# B&R Automation Studio project FactoryIO_Storage
Automation Studio 4.12.2.93; technology packages: mappView 5.16.1

## Configuration Config1

CPU PC_any, AutomationRuntime B4.93, Build 4.1.2, Vc V4.72.6

### Task classes (Cpu.sw)
```
Cyclic#1 (cycle 20000 us):
  _1000_SCTR <- _1000_SCTRL.prg
  _1100_CSYS <- _1100_CSYS.prg
  _1500_PPS <- _1500_PPS.prg
  _1700_HMI <- _1700_HMI.prg
  _1600_SSYS <- _1600_SSYS.prg
  _1400_SRS <- _1400_SRS.prg
  _1300_CS2 <- _1300_CS2.prg
  _1200_CS1 <- _1200_CS1.prg
Binaries: udbdef, FWRules, TCData, sysconf, Role, User, iomap, ashwd, asfw, arconfig, ashwac
Libraries: Library, runtime, astime, asieccon
```

### Hardware
```
OpcUa_any : OpcUa_any v1.0.0.1  [ETH1 -> PC.IF3 [Cable Type=PowerlinkCable, Length=10, Version=1.0.0.3]]
  ServerEndpointUrl = opc.tcp://127.0.0.1:48020
PC : PC_any v1.1.1.0 (OrderNumber=PC)
  ConfigurationID = FactoryIO_Storage_Config1
  Cyclic1Duration = 20000
  FileDevice1
  FileDeviceName1 = USER
  FileDevicePath1 = USER_PATH
  ActivateOpcUa = 1
  OpcUaInformationModels_PV_Version = 1
```

## Logical view

Binary libraries used (declarations not repeated): operator, runtime, astime, AsIecCon

### Global.var - Global variables
```iecst
VAR
	Gv : UDT_Global;
	Opc : UDT_Opc;
END_VAR
```

### Package Logical/Libraries - Global libraries

### Library Logical/Libraries/Library (IEC)

#### Modules.typ - Exported data types
```iecst
TYPE
	UDT_StorageController : 	STRUCT
		Dummy : BOOL;
	END_STRUCT;
	UDT_ControlSystem : 	STRUCT
		Dummy : BOOL;
	END_STRUCT;
	UDT_ConveyorInfeedSystem : 	STRUCT
		ReadyForOffload : BOOL;
	END_STRUCT;
	UDT_ConveyorOutfeedSystem : 	STRUCT
		ReadyForOnload : BOOL;
	END_STRUCT;
	UDT_StorageRackSystem : 	STRUCT
		Dummy : BOOL;
	END_STRUCT;
	UDT_HMI : 	STRUCT
		Dummy : BOOL;
	END_STRUCT;
	UDT_PickAndPlaceSystem : 	STRUCT
		Offloading : UDT_Sequence;
		Loading : UDT_Sequence;
	END_STRUCT;
	UDT_SafetySystem : 	STRUCT
		SafetyStop : BOOL;
		ControlledStop : BOOL;
	END_STRUCT;
END_TYPE
```

#### Library.fun - Exported functions and function blocks
```iecst
{REDUND_ERROR} FUNCTION_BLOCK FB_Loader (*TODO: Add your comment here*) (*$GROUP=User,$CAT=User,$GROUPICON=User.png,$CATICON=User.png*)
	VAR_INPUT
		in_xLimitRight : {REDUND_UNREPLICABLE} BOOL;
		in_xLimitLeft : {REDUND_UNREPLICABLE} BOOL;
		in_xLimitMiddle : {REDUND_UNREPLICABLE} BOOL;
		in_xInterlock : {REDUND_UNREPLICABLE} BOOL;
		in_xMovingX : {REDUND_UNREPLICABLE} BOOL;
		in_xMovingZ : {REDUND_UNREPLICABLE} BOOL;
		in_rZActualPos : REAL;
		in_rXActualPos : REAL;
		in_rLoadDeltaZ : REAL;
		in_xLoadRightReq : BOOL;
		in_xLoadLeftReq : BOOL;
		in_xUnloadRightReq : BOOL;
		in_xUnloadLeftReq : BOOL;
	END_VAR
	VAR_OUTPUT
		out_sStatus : {REDUND_UNREPLICABLE} UDT_Sequence;
		out_xForksLeftOrder : BOOL;
		out_xForksRightOrder : BOOL;
		out_rXSetPoint : REAL;
		out_rZSetPoint : REAL;
		out_xLoaded : BOOL;
	END_VAR
	VAR
		OperateRight : BOOL;
		OperateLeft : BOOL;
		Unload : BOOL;
		Load : BOOL;
		v_InPosition : BOOL;
		v_LoadSequence : DINT;
	END_VAR
END_FUNCTION_BLOCK

{REDUND_ERROR} FUNCTION_BLOCK FB_Crane (*TODO: Add your comment here*) (*$GROUP=User,$CAT=User,$GROUPICON=User.png,$CATICON=User.png*)
	VAR_INPUT
		in_rXSetPointReq : REAL;
		in_rZSetPointReq : REAL;
		in_rZActualPos : REAL;
		in_rXActualPos : REAL;
		in_xInterlock : BOOL;
	END_VAR
	VAR_OUTPUT
		out_sStatus : {REDUND_UNREPLICABLE} UDT_Sequence;
		out_rXSetPoint : REAL;
		out_rZSetPoint : REAL;
	END_VAR
	VAR
		InPosition : BOOL;
		Interlock : BOOL;
		NewRequest : BOOL;
		PreviousXSetPoint : REAL;
		PreviousZSetPoint : REAL;
		FirstScan : BOOL;
	END_VAR
END_FUNCTION_BLOCK
```

#### OPC.typ
```iecst
TYPE
	UDT_OpcInput : 	STRUCT
		StorageController : UDT_StorageControllerInput;
		ControlSystem : UDT_ControlSystemInput;
		ConveyorInfeed : UDT_ConveyorInfeedInput;
		ConveyorOutfeed : UDT_ConveyorOutfeedInput;
		StorageRack : UDT_StorageRackSystemInput;
		PickAndPlace : UDT_PickAndPlaceSystemInput;
		Safety : UDT_SafetySystemInput;
		HMI : UDT_HMIInput;
	END_STRUCT;
	UDT_OpcOutput : 	STRUCT
		StorageController : UDT_StorageControllerOutput;
		ControlSystem : UDT_ControlSystemOutput;
		ConveyorInfeed : UDT_ConveyorInfeedOutput;
		ConveyorOutfeed : UDT_ConveyorOutfeedOutput;
		StorageRack : UDT_StorageRackSystemOutput;
		PickAndPlace : UDT_PickAndPlaceSystemOutput;
		SafetySystem : UDT_SafetySystemOutput;
		HMI : UDT_HMIOutput;
	END_STRUCT;
	UDT_StorageControllerInput : 	STRUCT
		Opc_IO_Factory_Reset : BOOL;
		Opc_IO_Factory_Running : BOOL;
		Opc_IO_Factory_Paused : BOOL;
	END_STRUCT;
	UDT_ControlSystemInput : 	STRUCT
		Opc_IO_StartButton : BOOL;
		Opc_IO_StopButton : BOOL;
		Opc_IO_ManualSwitch : BOOL;
		Opc_IO_AutoSwitch : BOOL;
	END_STRUCT;
	UDT_ConveyorInfeedInput : 	STRUCT
		Opc_IO_AtEntry : BOOL;
		Opc_IO_AtLoad : BOOL;
	END_STRUCT;
	UDT_ConveyorOutfeedInput : 	STRUCT
		Opc_IO_AtExit : BOOL;
		Opc_IO_AtUnload : BOOL;
	END_STRUCT;
	UDT_StorageRackSystemInput : 	STRUCT
		Dummy : BOOL;
	END_STRUCT;
	UDT_PickAndPlaceSystemInput : 	STRUCT
		Opc_IO_PosZ : REAL;
		Opc_IO_PosX : REAL;
		Opc_IO_MovingX : BOOL;
		Opc_IO_MovingZ : BOOL;
		Opc_IO_LeftLimitSwitch : BOOL;
		Opc_IO_RightLimitSwitch : BOOL;
		Opc_IO_MiddleLimitSwitch : BOOL;
	END_STRUCT;
	UDT_SafetySystemInput : 	STRUCT
		Opc_IO_EmergencyStop1 : BOOL;
	END_STRUCT;
	UDT_HMIInput : 	STRUCT
		Dummy : BOOL;
	END_STRUCT;
	UDT_StorageControllerOutput : 	STRUCT
		Dummy : BOOL;
	END_STRUCT;
	UDT_ControlSystemOutput : 	STRUCT
		Opc_IO_ResetLight : BOOL;
		Opc_IO_StopLight : BOOL;
		Opc_IO_StartLight : BOOL;
	END_STRUCT;
	UDT_ConveyorInfeedOutput : 	STRUCT
		Opc_IO_LoadingConveyor : BOOL;
		Opc_IO_EntryConveyor : BOOL;
	END_STRUCT;
	UDT_ConveyorOutfeedOutput : 	STRUCT
		Opc_IO_UnloadConveyor : BOOL;
		Opc_IO_ExitConveyor : BOOL;
	END_STRUCT;
	UDT_StorageRackSystemOutput : 	STRUCT
		Dummy : BOOL;
	END_STRUCT;
	UDT_PickAndPlaceSystemOutput : 	STRUCT
		Opc_IO_ForksRight : BOOL;
		Opc_IO_XAxisSetPoint : REAL;
		Opc_IO_ZAxisSetPoint : REAL;
		Opc_IO_ForksLeft : BOOL;
	END_STRUCT;
	UDT_SafetySystemOutput : 	STRUCT
		Dummy : BOOL;
	END_STRUCT;
	UDT_HMIOutput : 	STRUCT
		Dummy : BOOL;
	END_STRUCT;
END_TYPE
```

#### Global.typ
```iecst
TYPE
	UDT_Opc : 	STRUCT
		In : UDT_OpcInput;
		Out : UDT_OpcOutput;
	END_STRUCT;
	UDT_Global : 	STRUCT
		StorageController : UDT_StorageController;
		ControlSystem : UDT_ControlSystem;
		ConveyorIn : UDT_ConveyorInfeedSystem;
		ConveyorOut : UDT_ConveyorOutfeedSystem;
		StorageRackSystem : UDT_StorageRackSystem;
		HMI : UDT_HMI;
		PickAndPlaceSystem : UDT_PickAndPlaceSystem;
		SafetySystem : UDT_SafetySystem;
	END_STRUCT;
END_TYPE
```

#### States.typ
```iecst
TYPE
	TSystemState :
		(
		Initializing,
		Running,
		Error,
		Maintenance,
		SafetyStop
		);
END_TYPE
```

#### SubState.typ
```iecst
TYPE
	UDT_Sequence : 	STRUCT
		Error : BOOL;
		Idle : BOOL;
		InProgess : BOOL;
		Requested : BOOL;
	END_STRUCT;
END_TYPE
```

#### DataTypes.typ - not listed in the package file held
```iecst
TYPE
	UDT_XYZCoordinate : 	STRUCT
		X : REAL;
		Y : REAL;
		Z : REAL;
	END_STRUCT;

END_TYPE
```

#### GV.typ - not listed in the package file held
```iecst
TYPE
	UDT_Opc : 	STRUCT
		In : UDT_OpcInput;
		Out : UDT_OpcOutput;
	END_STRUCT;

	UDT_Global : 	STRUCT
		StorageController : UDT_StorageController;
		ControlSystem : UDT_ControlSystem;
		ConveyorIn : UDT_ConveyorInfeedSystem;
		ConveyorOut : UDT_ConveyorOutfeedSystem;
		StorageRackSystem : UDT_StorageRackSystem;
		HMI : UDT_HMI;
		PickAndPlaceSystem : UDT_PickAndPlaceSystem;
		SafetySystem : UDT_SafetySystem;
		Params: TParameters;
	END_STRUCT;

	UDT_StorageController : 	STRUCT
		Dummy : BOOL;
	END_STRUCT;
	UDT_ControlSystem : 	STRUCT
		Dummy : BOOL;
	END_STRUCT;
	UDT_ConveyorInfeedSystem : 	STRUCT
		ReadyForOffload : BOOL;
	END_STRUCT;
	UDT_ConveyorOutfeedSystem : 	STRUCT
		ReadyForOnload : BOOL;
	END_STRUCT;
	UDT_StorageRackSystem : 	STRUCT
		Dummy : BOOL;
		StoragePlaceRequest : BOOL;
		StoragePlaceAcknowledge: TStorageSlot;
		(*StorageRackMatrix : ARRAY[1..10, 1..10] OF TStorageSlot;*)
	END_STRUCT;
	UDT_HMI : 	STRUCT
		Dummy : BOOL;
	END_STRUCT;
	UDT_PickAndPlaceSystem : 	STRUCT
		Offloading : UDT_Sequence;
		Loading : UDT_Sequence;
		ActualPositionX: REAL;
		ActualPositionZ: REAL;

	END_STRUCT;
	UDT_SafetySystem : 	STRUCT
		SafetyStop : BOOL;
		ControlledStop : BOOL;
	END_STRUCT;

	TParameters : 	STRUCT
		StorageSizeX : INT;
		StorageSizeZ : INT;
		FirstSlotXPos : REAL;
		FirstSlotZPos : REAL;
		LastSlotXPos : REAL;
		LastSlotZPos : REAL;
	END_STRUCT;

END_TYPE
```

#### Sequence.typ - not listed in the package file held
```iecst
TYPE
	UDT_Sequence : 	STRUCT
		Error : BOOL;
		Idle : BOOL;
		InProgress : BOOL;
		Requested : BOOL;
	END_STRUCT;
	UDT_Sequencer : 	STRUCT
		OnEntryFlag : BOOL := TRUE;
		CurrentStep : INT := 0;
		NextStep : INT := 0;
	END_STRUCT;
END_TYPE
```

#### StorageUdts.typ - not listed in the package file held
```iecst
TYPE

	TCoordinate : STRUCT
		x : REAL;
		z : REAL;
	END_STRUCT;

	TBoxData : STRUCT
		id : STRING;
		weight : REAL;
		isvalid : BOOL;
	END_STRUCT;

	TStorageSlot : STRUCT
		number : INT;
		coordinate : TCoordinate;
		available : BOOL;
		box : TBoxData;
	END_STRUCT;
END_TYPE
```

#### FB_Crane.st - not listed in the package file held
```iecst
(* TODO: Add your comment here *)
FUNCTION_BLOCK FB_Crane
//MovX	REAL	FALSE	VAR_INPUT		FALSE	FALSE		 	 	 	 	48
//	MovY	REAL	FALSE	VAR_INPUT		FALSE	FALSE		 	 	 	 	49
//	Status	UDT_Sequence		VAR_OUTPUT		FALSE	FALSE		 	 	 	 	7
//	XSetPoint	REAL		VAR_OUTPUT		FALSE	TRUE		 	 	 	 	-1
//	ZSetPoint	REAL		VAR_OUTPUT		FALSE	TRUE		 	 	 	 	-1

	NewRequest := NOT(PreviousXSetPoint = in_rXSetPointReq AND PreviousZSetPoint = in_rZSetPointReq);

	IF FirstScan THEN
		FirstScan := FALSE;
		out_sStatus.Idle := TRUE;
		out_rXSetPoint := in_rXActualPos;
		out_rZSetPoint := in_rZActualPos;
	END_IF;

	IF NOT in_xInterlock THEN
		IF NewRequest THEN
			out_rXSetPoint := in_rXSetPointReq;
			out_rZSetPoint := in_rZSetPointReq;
			out_sStatus.InProgress := TRUE;
			out_sStatus.Idle := FALSE;
		END_IF;
	ELSE
		out_rXSetPoint := in_rXActualPos;
		out_rZSetPoint := in_rZActualPos;
	END_IF;

	InPosition := ABS(out_rXSetPoint-in_rXActualPos)<0.05 AND ABS(out_rZSetPoint-in_rZActualPos)<0.05;
	IF InPosition AND out_sStatus.InProgress THEN
		out_sStatus.InProgress := FALSE;
		out_sStatus.Idle := TRUE;
	END_IF;

	PreviousXSetPoint := in_rXSetPointReq;
	PreviousZSetPoint := in_rZSetPointReq;

END_FUNCTION_BLOCK
```

#### FB_Loader.st - not listed in the package file held
```iecst
(* TODO: Add your comment here *)
FUNCTION_BLOCK FB_Loader

	v_InPosition := NOT in_xMovingX AND NOT in_xMovingZ;

	Load := in_xLoadRightReq OR in_xLoadLeftReq;
	Unload := in_xUnloadLeftReq OR in_xUnloadRightReq;
	OperateLeft := in_xUnloadLeftReq OR in_xLoadLeftReq;
	OperateRight := in_xUnloadRightReq OR in_xLoadRightReq;

	IF NOT out_sStatus.InProgress AND NOT (in_xLoadRightReq OR in_xLoadLeftReq OR in_xUnloadLeftReq OR in_xUnloadRightReq) THEN
		v_LoadSequence := 0;
		out_sStatus.InProgress := FALSE;
		out_sStatus.Idle := TRUE;
		out_xForksLeftOrder := FALSE;
		out_xForksRightOrder := FALSE;
	END_IF;

	IF Load THEN
		CASE v_LoadSequence OF
			0:
				out_sStatus.InProgress := FALSE;
				out_sStatus.Idle := TRUE;
				out_xForksLeftOrder := FALSE;
				out_xForksRightOrder := FALSE;
				IF NOT out_xLoaded THEN
					v_LoadSequence := 1;

				END_IF;
			1:
				out_sStatus.InProgress := TRUE;
				out_rZSetPoint := in_rZActualPos - in_rLoadDeltaZ;
				v_LoadSequence := 2;
			2:
				IF v_InPosition THEN
					v_LoadSequence := 3;
				END_IF;
			3:

				IF OperateLeft THEN
					out_xForksLeftOrder := TRUE;
					IF in_xLimitLeft THEN
						v_LoadSequence := 4;
					END_IF;
				ELSIF OperateRight THEN
					out_xForksRightOrder := TRUE;
					IF in_xLimitRight THEN
						v_LoadSequence := 4;
					END_IF;
				END_IF;

			4:
				out_rZSetPoint := in_rZActualPos + in_rLoadDeltaZ*2;
				v_LoadSequence := 5;
			5:
				IF v_InPosition THEN
					v_LoadSequence := 6;
				END_IF;
			6:
				out_xForksLeftOrder := FALSE;
				out_xForksRightOrder := FALSE;
				IF in_xLimitMiddle THEN
					v_LoadSequence := 7;
				END_IF;
			7:
				out_rZSetPoint := in_rZActualPos - in_rLoadDeltaZ;
				v_LoadSequence := 8;
			8:
				IF v_InPosition THEN
					v_LoadSequence := 9;
				END_IF;
			9:
				out_xLoaded := TRUE;
				out_sStatus.InProgress := FALSE;
				out_sStatus.Idle := TRUE;
				v_LoadSequence := 0;
		END_CASE
	ELSIF Unload THEN
		CASE v_LoadSequence OF
			0:
				out_sStatus.InProgress := FALSE;
				out_sStatus.Idle := TRUE;
				out_xForksLeftOrder := FALSE;
				out_xForksRightOrder := FALSE;
				IF out_xLoaded THEN
					v_LoadSequence := 1;

				END_IF;
			1:
				out_sStatus.InProgress := TRUE;
				out_rZSetPoint := in_rZActualPos + in_rLoadDeltaZ;
				v_LoadSequence := 2;
			2:
				IF v_InPosition THEN
					v_LoadSequence := 3;
				END_IF;
			3:
				IF OperateRight THEN
					out_xForksRightOrder := TRUE;
					IF in_xLimitRight THEN
						v_LoadSequence := 4;
					END_IF;
				ELSIF OperateLeft THEN
					out_xForksLeftOrder := TRUE;
					IF in_xLimitLeft THEN
						v_LoadSequence := 4;
					END_IF;
				END_IF;
			4:
				out_rZSetPoint := in_rZActualPos - in_rLoadDeltaZ * 2;
				v_LoadSequence := 5;
			5:
				IF v_InPosition THEN
					v_LoadSequence := 6;
				END_IF;
			6:
				out_xForksLeftOrder := FALSE;
				out_xForksRightOrder := FALSE;
				IF in_xLimitMiddle THEN
					v_LoadSequence := 7;
				END_IF;
			7:
				out_rZSetPoint := in_rZActualPos + in_rLoadDeltaZ;
				v_LoadSequence := 8;
			8:
				IF v_InPosition THEN
					v_LoadSequence := 9;
				END_IF;
			9:
				out_xLoaded := FALSE;
				v_LoadSequence := 0;
		END_CASE
	END_IF

END_FUNCTION_BLOCK
```

- Visualisation Logical/mappView (not shown)

- OpcTag.opct (not shown)

- OpcProperties.opcp (not shown)

### Program Logical/_1000_SCTRL (IEC)

#### Variables.var - Local variables
```iecst
VAR
	in : UDT_;
END_VAR
```

#### Init.st - Init code
```iecst
PROGRAM _INIT
	(* Insert code here *)
	Gv.Params.StorageSizeX := 9;
	Gv.Params.StorageSizeZ := 6;
	Gv.Params.FirstSlotXPos :=1.435;
	Gv.Params.FirstSlotZPos := 0.55;
	Gv.Params.LastSlotXPos := 10;
	Gv.Params.LastSlotZPos := 9.05;

END_PROGRAM
```

#### _0000_States.st - Cyclic code
```iecst
PROGRAM _CYCLIC

END_PROGRAM
```

#### _Controller__.st - not listed in the package file held
```iecst
PROGRAM _CYCLIC

END_PROGRAM
```

### Program Logical/_1010_SCTRL (ANSIC)

#### WorkOrderHandler.cpp - Init, cyclic, exit code
```cpp
#include <bur/plctypes.h>

#ifdef _DEFAULT_INCLUDES
	#include <AsDefault.h>
#endif

// amount of memory to be allocated for heap storage must be specified for every ANSI C++ program with the bur_heap_size variable
unsigned long bur_heap_size = 0xFFFF;

void _INIT ProgramInit(void)
{
	// Insert code here

}

void _CYCLIC ProgramCyclic(void)
{
	// Insert code here

}

void _EXIT ProgramExit(void)
{
	// Insert code here

}
```

- Program Logical/_1100_CSYS (IEC) (no source held here)

### Program Logical/_1200_CS1 (IEC)

#### Variables.var - Local variables
```iecst
VAR
	OpcOut : UDT_ConveyorInfeedOutput;
	OpcIn : UDT_ConveyorInfeedInput;
	Gv : UDT_Global;
END_VAR
VAR CONSTANT
	STS_Idle : USINT := 0;
	STS_Transfer : USINT := 1;
	STS_WaitForOffload : USINT := 2;
END_VAR
VAR
	v_CurrentState : USINT := 0;
	v_BoxAtEntry : BOOL;
	v_BoxAtLoad : BOOL;
	v_OffloadingActive : BOOL;
	v_ReadyToOffload : BOOL;
	v_EntryConveyorRunOrder : BOOL;
	v_LoadingConveyorRunOrder : BOOL;
END_VAR
```

#### Types.typ - Local data types
```iecst
TYPE
	States :
		(
		Idle,
		TransferToLoading,
		ReadyForOffload
		);
END_TYPE
```

#### _0100_Controller.st - Cyclic code
```iecst
PROGRAM _CYCLIC

	// INPUTS
		// OPC Inputs
	v_BoxAtEntry := NOT Opc.In.ConveyorInfeed.Opc_IO_AtEntry;
	v_BoxAtLoad := NOT Opc.In.ConveyorInfeed.Opc_IO_AtLoad;

    	// Module Inputs
	v_OffloadingActive := Gv.PickAndPlaceSystem.Offloading.InProgess;

	CASE v_CurrentState OF
		STS_Idle:
			IF v_BoxAtEntry AND NOT v_BoxAtLoad AND NOT v_OffloadingActive THEN
				v_CurrentState := STS_Transfer;
			END_IF;
		STS_Transfer:
			v_EntryConveyorRunOrder := TRUE;
			v_LoadingConveyorRunOrder := TRUE;
			IF v_BoxAtLoad THEN
				v_CurrentState := STS_WaitForOffload;
			END_IF;
		STS_WaitForOffload:
			IF NOT v_BoxAtLoad AND NOT v_OffloadingActive THEN
				v_ReadyToOffload := FALSE;
				v_CurrentState := STS_Idle;
			END_IF;
	END_CASE;

	IF v_CurrentState = STS_Idle THEN

		v_EntryConveyorRunOrder := FALSE;
		v_LoadingConveyorRunOrder := FALSE;

	ELSIF v_CurrentState = STS_Transfer THEN

		v_EntryConveyorRunOrder := TRUE;
		v_LoadingConveyorRunOrder := TRUE;

	ELSIF v_CurrentState = STS_WaitForOffload THEN

		v_ReadyToOffload := TRUE;
		v_EntryConveyorRunOrder := FALSE;
		v_LoadingConveyorRunOrder := FALSE;

	ELSE
		// State error
	END_IF;

	// OUTPUTS
		// OPC outputs
	Opc.Out.ConveyorInfeed.Opc_IO_EntryConveyor := v_EntryConveyorRunOrder;
	Opc.Out.ConveyorInfeed.Opc_IO_LoadingConveyor := v_LoadingConveyorRunOrder;

		// Module output
	Gv.ConveyorIn.ReadyForOffload := v_ReadyToOffload;

END_PROGRAM
```

#### _0000_States.st - not listed in the package file held
```iecst
PROGRAM _CYCLIC
	in := Opc.In.ConveyorInfeed;

END_PROGRAM
```

- Program Logical/_1300_CS2 (IEC) (no source held here)

### Program Logical/_1400_SRS (IEC)

#### Variables.var - Local variables
```iecst
VAR
	v_StorageTaken : ARRAY[1..8, 1..10] OF BOOL;

	v_StorageCoordinates : ARRAY[1..8, 1..10] OF BOOL;
	StorageRack : BOOL;
	NextAvailableX : BOOL;
	NextAvailableZ : BOOL;

END_VAR

VAR CONSTANT

END_VAR
```

#### _0100_Controller.st - Cyclic code
```iecst
PROGRAM _CYCLIC

END_PROGRAM
```

### Program Logical/_1410_SRS (ANSIC)

#### Cyclic.cpp
```cpp
#include <bur/plctypes.h>

#ifdef _DEFAULT_INCLUDES
#include <AsDefault.h>
#endif

unsigned long bur_heap_size = 0xFFFF; // Define heap size for dynamic memory allocation

// Define a struct to represent coordinates
struct Coordinates {
	int x;
	int z;
};

class RisingEdge {
private:
    bool lastState; // Variable to keep track of the last state of the signal

public:
    // Constructor
    RisingEdge() : lastState(false) {} // Initialize lastState to false

    // Function to check for a rising edge
    bool detect(bool currentState) {
        bool isRisingEdge = !lastState && currentState; // Check if the last state was false and current state is true
        lastState = currentState; // Update the last state to the current state
        return isRisingEdge; // Return true if a rising edge is detected, otherwise false
    }
};

// Define a class to represent the storage rack
class StorageRack {
	public:
	static const int width = 9;
	static const int depth = 6;
	bool slots[depth][width]; // true if available, false if occupied

	// Constructor to initialize all slots to available
	StorageRack() {
		for(int z = 0; z < depth; ++z) {
			for(int x = 0; x < width; ++x) {
				slots[z][x] = true;
			}
		}
	}

	// Function to find the closest available slot to a given position
	Coordinates findClosestAvailable(int inputX, int inputZ) {
		int minDistance = width * depth; // Initialize with maximum possible distance
		Coordinates closestSlot = {-1, -1}; // Initialize to an invalid position

		for(int z = 0; z < depth; ++z) {
			for(int x = 0; x < width; ++x) {
				if(slots[z][x]) { // Slot is available
					int distance = 0; //abs(inputX - x) + abs(inputZ - z); // Calculate Manhattan distance
					if(distance < minDistance) {
						closestSlot.x = x;
						closestSlot.z = z;
						minDistance = distance;
					}
				}
			}
		}
		return closestSlot; // Return the coordinates of the closest slot
	}

};

StorageRack myRack; // Instantiate the storage rack
RisingEdge risingEdge;

void _CYCLIC ProgramCyclic(void)
{

	//if(risingEdge.detect(Gv.StorageRackSystem.RequestCoordinates)) {
					// Rising edge detected, insert the logic to handle a rising edge event
	//}

}
```

### Program Logical/_1500_PPS (IEC)

#### Variables.var - Local variables
```iecst
VAR
	v_LeftLimitSwitch : BOOL;
	v_MiddleLimitSwitch : BOOL;
	v_RightLimitSwitch : BOOL;
	v_MovingX : BOOL;
	v_MovingZ : BOOL;
	v_ActualPositionX : REAL;
	v_ActualPositionZ : REAL;
	v_ForksLeftExtendOrder : BOOL;
	v_ForksRightExtendOrder : BOOL;
	v_CraneXAxisSetPoint : REAL;
	v_CraneZAxisSetPoint : REAL;
	v_InfeedPickupAndStoreReq : BOOL;
	test_rPosXReq : REAL;
	test_rPosZReq : REAL;
	test_xLoadLeft : BOOL;
	test_xUnloadRight : BOOL;
	test_xLoadRight : BOOL;
	test_xUnloadLeft : BOOL;
	PAR_HomeX : REAL;
	PAR_HomeZ : REAL;
	PAR_NbrOfTiers : DINT;
	PAR_NbrOfRows : DINT;
	PAR_FirstBayPosX : REAL;
	PAR_FirstBayPosZ : REAL;
	PAR_LastBayPosX : REAL;
	PAR_LastBayPosZ : REAL;
	PAR_LoadOffLoadZDelta : REAL;
	fb_Loader : FB_Loader;
	fb_Crane : FB_Crane;
	STS_Load_Left : {REDUND_UNREPLICABLE} DINT := 1;
	STS_Load_Right : {REDUND_UNREPLICABLE} DINT := 2;
	STS_MoveToTarget : {REDUND_UNREPLICABLE} DINT := 3;
	STS_Unload : {REDUND_UNREPLICABLE} DINT := 4;
	FirstScan : BOOL;
	STS_PickAndPlace : UDT_Sequencer;
	STS_Offload : INT;
	STS_Store : INT;
	STS_Load : INT;
v_xTest : BOOL;
END_VAR
VAR CONSTANT
	STS_Init : INT := 0;
	STS_Idle : INT := 1;
	STS_LoadFromConveyor : INT := 2;
	STS_LoadFromStorage : INT := 3;
	STS_OffloadInStorage : INT := 4;
	STS_OffloadOnConveyour : INT := 5;
END_VAR
VAR
	SEQ_LoadFromConveyor : UDT_Sequencer;
	v_StorageFull : BOOL;
	SQS_OffloadInStorage : UDT_Sequencer;
END_VAR
```

#### Init.st - Init code
```iecst
PROGRAM _INIT
	(* Insert code here *)

	PAR_HomeX := 0.000;
	PAR_HomeZ := 0.180;

	PAR_FirstBayPosX := 01.425;
	PAR_FirstBayPosZ := 00.550;

	PAR_LastBayPosX := 10.000;
	PAR_LastBayPosZ := 09.050;

	PAR_NbrOfTiers := 6;
	PAR_NbrOfRows := 9;

	PAR_LoadOffLoadZDelta := 0.100;

END_PROGRAM
```

#### _0100_Controller.st - Cyclic code
```iecst
PROGRAM _CYCLIC

	// INPUTS
		// OPC
	v_LeftLimitSwitch 		:= Opc.In.PickAndPlace.Opc_IO_LeftLimitSwitch;
	v_MiddleLimitSwitch 	:= Opc.In.PickAndPlace.Opc_IO_MiddleLimitSwitch;
	v_RightLimitSwitch 		:= Opc.In.PickAndPlace.Opc_IO_RightLimitSwitch;
	v_MovingX				:= Opc.In.PickAndPlace.Opc_IO_MovingX;
	v_MovingY				:= Opc.In.PickAndPlace.Opc_IO_MovingZ;
	v_PositionX				:= Opc.In.PickAndPlace.Opc_IO_PosX;
	v_PositionZ				:= Opc.In.PickAndPlace.Opc_IO_PosZ;

		// GLOBAL

	// SEQUENCER
	CASE v_CurrentState OF
		STS_Idle:
			IF TRUE THEN
				v_CurrentState := STS_Transfer;
			END_IF;

		STS_WaitForLoad:
			IF TRUE THEN
				v_CurrentState := STS_Transfer;
			END_IF;

		STS_Load:
			IF TRUE THEN
				v_CurrentState := STS_Transfer;
			END_IF;

		STS_MoveToTarget:
			IF TRUE THEN
				v_CurrentState := STS_Transfer;
			END_IF;

		STS_Unload:
			IF TRUE THEN
				v_CurrentState := STS_Transfer;
			END_IF;
	END_CASE;

	// ACTIONS

	// OUTPUTS
		// OPC
	Opc.Out.PickAndPlace.Opc_IO_ForksLeft := v_ForksLeftExtendOrder;
	Opc.Out.PickAndPlace.Opc_IO_ForksRight := v_ForksRightExtendOrder;

	Opc.Out.PickAndPlace.Opc_IO_XAxisSetPoint := v_CraneXAxisSetPoint;
	Opc.Out.PickAndPlace.Opc_IO_ZAxisSetPoint := v_CraneZAxisSetPoint;
		// GLOBAL
	//Storage Full

END_PROGRAM
```

### Variables.var
```iecst
VAR
	var_StartReq : BOOL;
	var_StartOrder : BOOL;
	var_Counter : DINT;
	var_StartReqPreviousState : BOOL;
END_VAR
```

Listed in the project but not available here: Logical/Global.typ, Logical/Libraries/Library/Constants.var, Logical/_1000_SCTRL/Types.typ, Logical/_1000_SCTRL/Exit.st, Logical/_1010_SCTRL/Types.typ, Logical/_1010_SCTRL/Variables.var, Logical/_1100_CSYS/Variables.var, Logical/_1100_CSYS/_0000_States.st, Logical/_1100_CSYS/Init.st, Logical/_1100_CSYS/Exit.st, Logical/_1100_CSYS/Types.typ, Logical/_1200_CS1/Init.st, Logical/_1200_CS1/Exit.st, Logical/_1300_CS2/Init.st, Logical/_1300_CS2/Exit.st, Logical/_1300_CS2/Types.typ, Logical/_1300_CS2/Variables.var, Logical/_1300_CS2/_0000_States.st, Logical/_1400_SRS/Init.st, Logical/_1400_SRS/Exit.st, Logical/_1400_SRS/Types.typ, Logical/_1500_PPS/Exit.st, Logical/_1500_PPS/Types.typ, Logical/_1600_SSYS, Logical/_1700_HMI
